{attribute 'linkalways'} 
{attribute 'no_explicit_call' := 'This FB is a CLASS and must be accessed using methods or properties'}
{attribute 'enable_dynamic_creation'}
FUNCTION_BLOCK FINAL MIN_WORD EXTENDS Node
VAR
	in1 : _WORD(0);
	in2 : _WORD(0);
	out : _WORD(0);
END_VAR

METHOD PUBLIC Clone : I_Node
VAR
	pNode : POINTER TO MIN_WORD;
END_VAR
pNode := __NEW(MIN_WORD);
Clone := pNode^;
END_METHOD

METHOD FB_init : BOOL
VAR_INPUT
	bInitRetains : BOOL; // if TRUE, the retain variables are initialized (warm start / cold start)
	bInCopyCode : BOOL;  // if TRUE, the instance afterwards gets moved into the copy code (online change)
END_VAR
AddInput('in1',THIS^.in1);
AddInput('in2',THIS^.in2);
AddOutput('out', THIS^.out);
END_METHOD

METHOD PROTECTED OnExecute
VAR
END_VAR
out.Value := MIN(in1.Value, in2.Value);
END_METHOD

END_FUNCTION_BLOCK

(* stored: Version 1.1.0.1, ProductVersion 3.1.4024.15
   POU MIN_WORD: Id {1f7b4bff-7e76-48c5-b847-3e8e36a2f966}, SpecialFunc None
   Folder Constructor: Id {64b75dbe-82dc-4c92-a1ae-cf3ec6b7bcac}
   Method Clone: Id {eccaf5e3-1696-4b5e-9e24-3a9b103323b9}
   Method FB_init: Id {79baf21d-e4d4-46da-b925-955d32b1b4cb}
   Method OnExecute: Id {d75bc0ab-fc31-42f0-b867-86b3555d7f19} *)
